{attribute addProperty BoxType "AX5021-0000-0002-0002"}
{attribute addProperty Id "Master_control_wordAT %Q*UINT162"}
{attribute addProperty CRC "2179244868"}
{attribute addProperty SizeInBites "16"}
{attribute addProperty SizeInBytes "2"}
TYPE MDT_81E4A344 :
STRUCT
	{attribute addProperty Name "Master_control_word"}
	Master_control_word AT %Q* : UINT;
END_STRUCT
END_TYPE

(* stored: Version 1.2.0.0, ProductVersion 3.1.4024.9
   DUT MDT_81E4A344: Id {5489c473-aca6-4f38-a6ff-1ea795fc54cf} *)
